FUNCTION_BLOCK FB_ControlElement5 EXTENDS FB_BaseControlElement IMPLEMENTS ITF_ControlElement5
VAR
	
	itfsenStart			: ITF_IOSensor;
	itfsenEnd			: ITF_IOSensor;	
END_VAR

METHOD FB_init : BOOL
VAR_INPUT
	bInitRetains : BOOL; // if TRUE, the retain variables are initialized (warm start / cold start)
	bInCopyCode : BOOL;  // if TRUE, the instance afterwards gets moved into the copy code (online change)
	itfsenStart			: ITF_IOSensor;
	itfsenEnd			: ITF_IOSensor;	
	
END_VAR
THIS^.itfsenStart					:= itfsenStart;
THIS^.AddComponent (itfComponent	:= itfsenStart);
THIS^.SetText (eLocation 			:= E_BaseLocation.pl, wsDescription := "Nazwa komponentu 1 pl");
THIS^.SetText (eLocation 			:= E_BaseLocation.en, wsDescription := "Nazwa komponentu 1 en");
THIS^.SetText (eLocation 			:= E_BaseLocation.de, wsDescription := "Nazwa komponentu 1 de");
THIS^.itfsenStart.SetName (stName	:= THIS^.GetTexts ());

THIS^.itfsenEnd						:= itfsenEnd;
THIS^.AddComponent (itfComponent	:= itfsenEnd);
THIS^.SetText (eLocation 			:= E_BaseLocation.pl, wsDescription := "Nazwa komponentu 2 pl");
THIS^.SetText (eLocation 			:= E_BaseLocation.en, wsDescription := "Nazwa komponentu 2 en");
THIS^.SetText (eLocation 			:= E_BaseLocation.de, wsDescription := "Nazwa komponentu 2 de");
THIS^.itfsenEnd.SetName (stName	:= THIS^.GetTexts ());
END_METHOD

END_FUNCTION_BLOCK

(* stored: Version 1.1.0.1, ProductVersion 3.1.4024.15
   POU FB_ControlElement5: Id {5a573246-27e9-4d44-ba35-7c33ce8d53d7}, SpecialFunc None
   Method FB_init: Id {6bd46216-6e61-4006-b610-fa2b62b42c21} *)
